{attribute 'qualified_only'}
{attribute 'TcHmiSymbol.AddSymbol'}
VAR_GLOBAL
    // Ring buffer of the most recent log entries the PLC has produced.
    // The Python bridge polls nWriteIdx via ADS and drains new slots.
    //   write slot at any moment = (nWriteIdx MOD 256)
    //   overflow detected when (nWriteIdx - lastReadIdx) > 256
    aLog        : ARRAY[0..255] OF ST_LogEntry;

    // Monotonic write counter (never wraps in practice — UDINT overflows
    // after 2^32 writes ≈ 4.3 billion, decades even at 1 kHz logging).
    nWriteIdx   : UDINT;

    // Global mute for PLC-side logging. When FALSE, F_LogEvent early-returns
    // without writing to aLog or aRecent. HMI Logs page binds this.
    bLogEnabled : BOOL := TRUE;

    // Runtime toggle for DEBUG severity. F_LogEvent drops DBG entries
    // when this is FALSE. Operator can flip it from the HMI without a
    // rebuild. HMI ToggleSwitch on the Robot page binds here.
    bDebugMode  : BOOL := FALSE;

    // Newest-first mirror of the last 20 entries. F_LogEvent shifts the
    // slots down and writes aRecent[0] on every accepted call, so the HMI
    // Logs page can bind aRecent[0..19] directly in display order.
    // aRecent[0] is the newest entry.
    aRecent     : ARRAY[0..19] OF ST_LogEntry;

    // Wall-clock HH:MM:SS, refreshed once a second by MAIN from
    // FB_LocalSystemTime, and copied into every entry by F_LogEvent.
    // It lives here rather than inside F_LogEvent because a FUNCTION cannot
    // own the FB instance FB_LocalSystemTime needs — functions are stateless,
    // so the cyclic tick has to happen in a POU that has one.
    // Reads '--:--:--' until the time source reports valid, so a panel with
    // an unset RTC shows that plainly instead of a plausible wrong time.
    sNow        : STRING(8) := '--:--:--';

    // Wall-clock date YYYY-MM-DD, refreshed by MAIN section 0a alongside sNow
    // but only when the DAY rolls over. Exists because filenames need a date
    // and sNow is HH:MM:SS only.
    //
    // Reads '0000-00-00' until the time source reports valid, and the writer
    // treats that as "no date" and falls back to flower-nodate-NNN.csv rather
    // than building a filename out of it. An unset panel RTC is a real
    // condition here, not a hypothetical -- sNow already has the same guard.
    // The sortable YYYY-MM-DD order is load-bearing for Phase 3: retention
    // deletes oldest-by-NAME, which is only correct because these sort
    // chronologically.
    sToday      : STRING(10) := '0000-00-00';

    // Durable CSV log status -- Phase 1 of docs/plans/log-csv-file.md.
    // VOLATILE on purpose (GVL_Log is plain VAR_GLOBAL): the config persists,
    // the status must not. A restored byte count or a stale FAILED with a
    // plausible error string would describe a file this runtime never opened.
    stLogFile   : ST_HmiLogFile;

    // ---------------------------------------------------------------- //
    // THROWAWAY -- Phase 0 gate of docs/plans/log-csv-file.md.
    // DELETE this whole block together with FB_LogFileSpike and
    // ST_LogFileProbe once the probe has answered. It is scaffolding for
    // deciding whether the CSV logger can be built, not part of it.
    //
    // Deliberately VOLATILE (GVL_Log is plain VAR_GLOBAL): a probe result is
    // evidence about one boot of one target, and persisting it would let a
    // stale PASS from the bench PC be read later as if it came from the panel.
    // The real logger's config goes in GVL_HmiPersistent in Phase 1 -- that
    // one has to survive, for the same reason sRobotHost does.
    // ---------------------------------------------------------------- //

    // Set TRUE (ADS or VISU) to run one sweep. FB_LogFileSpike edge-detects it
    // and self-clears, so it cannot re-run every scan and append six lines
    // per scan to whichever candidates work.
    bLogFileProbeRun   : BOOL;
    bLogFileProbeBusy  : BOOL;
    bLogFileProbeDone  : BOOL;

    // Set TRUE to DELETE the probe files from all six candidate locations.
    // Added 2026-08-10 because the first sweep left flower-spike.csv in four
    // places on the panel -- including, via PATH_BOOTPATH, next to
    // Port_851.bootdata -- and the probe had no way to remove them. A tool that
    // writes to a filesystem nobody can browse must be able to clean up after
    // itself. Same edge-trigger and self-clear as the run flag.
    bLogFileProbeCleanup : BOOL;

    // How many of the six candidates fully worked, and the index of the first
    // that did. -1 means none -- read that as "the file blocks or the target
    // are the problem", not "try a different path".
    nLogFileProbeOk    : INT;
    iLogFileProbeFirst : INT := -1;

    // One row per candidate. aLogFileProbe[i].sPathName is the value to carry
    // into stLogFileCfg.sDir in Phase 1, so it records what was actually
    // passed to FB_FileOpen rather than something reconstructed from it.
    aLogFileProbe      : ARRAY[1..6] OF ST_LogFileProbe;

    // NOTE stBridgeCfg / ST_LogBridgeCfg used to live here and are GONE
    // (2026-08-07). The field existed solely so the retired
    // RobotBridge/log_pump.py could publish its own logger configuration for an
    // HMI to render. The bridge was retired 2026-07-26 and nothing wrote the
    // struct after that, so it read as empty strings and zeros and made a
    // shipped FlowerPyHmi page render a visibly blank block. Removed from
    // FlowerPyHmi first, then from here -- that order matters, because deleting
    // the symbol while the poller still asks for it makes read_many log
    // "dropping N unresolvable symbol(s)", which looks like a real fault.
END_VAR

(* stored: Version 1.1.0.1, ProductVersion 3.1.4026.18
   GVL GVL_Log: Id {364bb45e-a498-4daa-a47c-ed8ea18daa8b} *)
